// TIA Portal V18 export
ORGANIZATION_BLOCK "Main"   // OB1, LAD, ProgramCycle
TITLE = "Main Program Sweep (Cycle)"
{ S7_Optimized_Access := 'TRUE' }
// stored: SetENOAutomatically false
   VAR_INPUT
      Initial_Call : Bool;   // Initial call of this OB
      Remanence : Bool;   // =True, if remanent data are available
   END_VAR
BEGIN

REGION Network 1
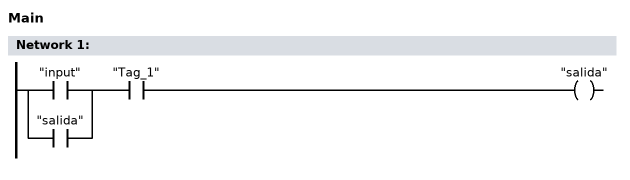
   RUNG wire#powerrail
      Contact( "input" )
      wire#w1
      Contact( "Tag_1" )
      Coil( "salida" )
   END_RUNG
   RUNG wire#powerrail
      Contact( "salida" )
   END_RUNG wire#w1
   // the same network as SCL:
   "salida" := ("input" OR "salida") AND "Tag_1";
END_REGION
END_ORGANIZATION_BLOCK
